// TwinCAT 3 PLC project ErrorTracker
// ProgramVersion: 3.1.4023.0
// libraries:
//   Tc2_Standard, * (Beckhoff Automation GmbH)
//   Tc2_System, * (Beckhoff Automation GmbH)
//   Tc2_Utilities, * (Beckhoff Automation GmbH)
//   Tc3_Module, * (Beckhoff Automation GmbH)
// project tree:
//   Diag/ CheckBounds.TcPOU, CheckDivDInt.TcPOU, CheckDivLInt.TcPOU, CheckDivLReal.TcPOU, CheckDivReal.TcPOU, CheckLRangeSigned.TcPOU, CheckLRangeUnsigned.TcPOU, CheckPointer.TcPOU, CheckRangeSigned.TcPOU, CheckRangeUnsigned.TcPOU, E_ErrType.TcDUT, FB_UdintTrig.TcPOU, G_Diag.TcGVL, prgDiag.TcPOU, stErrType.TcDUT, Visu_Diag.TcVIS
//   / GlobalTextList.TcGTLO, PlcTask.TcTTO, Visualization Manager.TcVMO (not stored)
//   POUs/ MAIN.TcPOU
// real-time tasks:
//   TASK PlcTask: cycle T#10ms, priority 20, ADS port 350
// I/O:
//   DEVICE Device 1 (EtherCAT) (disabled), AmsNetId 5.80.91.146.2.1
//     Term 1 (EK1100) [EK1100 EtherCAT Coupler (2A E-Bus)]
//       Term 2 (EL2008) [EL2008 8Ch. Dig. Output 24V, 0.5A]
// variable links:
//   ErrorTracker/ErrorTracker Instance <-> Device 1 (EtherCAT)
//     PlcTask Inputs/prgDiag.uiECatState <-> Inputs/DevState

CONFIGURATION ErrorTracker
    RESOURCE PLC ON TwinCAT3
        TASK PlcTask(INTERVAL := T#10ms, PRIORITY := 20);
        PROGRAM MAIN WITH PlcTask : MAIN;
    END_RESOURCE
END_CONFIGURATION

// ---- Diag/E_ErrType.TcDUT
{attribute 'qualified_only'}
{attribute 'strict'}
TYPE E_ErrType :
(
	eFirStErr,
	eCheckBoundsErr,
	eCheckDivDint,
	eCheckDivLint,
	eCheckDivReal,
	eCheckRange,
	eCheckPointer,
	eEtherCATErr,
	eRuntimeErr,
	eLastErr
);
END_TYPE

// ---- Diag/stErrType.TcDUT
TYPE stErrType :
STRUCT
	horario:DT;
	eErrType:E_ErrType;
END_STRUCT
END_TYPE

// ---- Diag/G_Diag.TcGVL
{attribute 'qualified_only'}
VAR_GLOBAL PERSISTENT
	uiCheckBound:UDINT;
	uiCheckDivDint:UDINT;
	uiCheckDivLint:UDINT;
	uiCheckDivReal:UDINT;
	uiCheckRange:UDINT;
	uiCheckPointer:UDINT;
	uiErrEtherCAT:UDINT;
	uiRuntimeErr:UDINT;
	aErrList:ARRAY[1..uiMaxNumOfErr] OF stErrType;
	uiECatState:UINT;
END_VAR
VAR_GLOBAL CONSTANT
	uiMaxNumOfErr:UINT:=100;
END_VAR

// ---- POUs/MAIN.TcPOU
PROGRAM MAIN
VAR
	i1,i2:INT;
	i3:INT:=5;
END_VAR
//An UPS is necessary to save the persistent Data, if it's not available other options are also possible, such as:
//Save to retain data / text files/Databases or simple use the FB_WritePersistentData and soon as a new error occur to make sure it's gonna be persistent
//Note : leaving Checks activated on a running machine can have negative effects on the performance
//As you find out what's the problem you should also remove checks from your code

//Here we call the program which handles the diagnosis
//
prgDiag();

i1:=i2/i3;

END_PROGRAM

// ---- Diag/prgDiag.TcPOU
PROGRAM prgDiag
VAR
	aErrTrig:ARRAY[E_ErrType.eFirStErr..E_ErrType.eLastErr] OF FB_UdintTrig;
	taskInfo:PlcTaskSystemInfo;
	
	horaAtual: DT;
	uiECatState AT %I*:UINT;
	localTyme:FB_LocalSystemTime;
	trigECAT:R_TRIG;
	timeStartup: TON := (PT := TIME#2S0MS);
	
END_VAR

timeStartup(IN:= TRUE);

IF NOT timeStartup.Q THEN
	RETURN;
END_IF

localTyme(
	sNetID:= '', 
	bEnable:= TRUE, 
	dwCycle:= , 
	dwOpt:= , 
	tTimeout:= , 
	bValid=> , 
	systemTime=> , 
	tzID=> );


taskInfo := _TaskInfo[1];

aErrTrig[E_ErrType.eCheckBoundsErr](uiIn:=G_Diag.uiCheckBound);
aErrTrig[E_ErrType.eCheckDivDint](uiIn:=G_Diag.uiCheckDivDint);
aErrTrig[E_ErrType.eCheckDivLint](uiIn:=G_Diag.uiCheckDivLint);
aErrTrig[E_ErrType.eCheckDivReal](uiIn:=G_Diag.uiCheckDivReal);
aErrTrig[E_ErrType.eCheckRange](uiIn:=G_Diag.uiCheckRange);
aErrTrig[E_ErrType.eCheckPointer](uiIn:=G_Diag.uiCheckPointer);


horaAtual:=SYSTEMTIME_TO_DT(localTyme.systemTime);	//==> colocar a hora do sistema aqui 
{Region "Checks"}
IF aErrTrig[E_ErrType.eCheckBoundsErr].bOut THEN
	M_InsertOnList(eErrInsert:=E_ErrType.eCheckBoundsErr , hora:=horaAtual );
END_IF
IF aErrTrig[E_ErrType.eCheckDivDint].bOut THEN
	M_InsertOnList(eErrInsert:=E_ErrType.eCheckDivDint , hora:=horaAtual );	
END_IF
IF aErrTrig[E_ErrType.eCheckDivLint].bOut THEN
	M_InsertOnList(eErrInsert:= E_ErrType.eCheckDivLint, hora:=horaAtual );	
END_IF
IF aErrTrig[E_ErrType.eCheckDivReal].bOut THEN
	M_InsertOnList(eErrInsert:= E_ErrType.eCheckDivReal, hora:=horaAtual );	
END_IF
IF aErrTrig[E_ErrType.eCheckRange].bOut THEN
	M_InsertOnList(eErrInsert:=E_ErrType.eCheckRange , hora:=horaAtual );	
END_IF
IF aErrTrig[E_ErrType.eCheckPointer].bOut THEN
	M_InsertOnList(eErrInsert:= E_ErrType.eCheckPointer, hora:=horaAtual );	
END_IF
{endregion}

{Region "EtherCAT"}
	trigECAT(CLK:=uiECatState <> 0);
	IF trigECAT.Q THEN
		 M_InsertOnList(eErrInsert:= E_ErrType.eEtherCATErr, hora:=horaAtual );
		 G_Diag.uiECatState:=uiECatState;
	END_IF
{endregion}

{Region "Runtime"}
	IF taskInfo.CycleTimeExceeded THEN
		G_Diag.uiRuntimeErr:=G_Diag.uiRuntimeErr+1;
		M_InsertOnList(eErrInsert:= E_ErrType.eRuntimeErr, hora:=horaAtual );	
	END_IF
{endregion}

METHOD M_InsertOnList : BOOL
VAR_INPUT
	eErrInsert:E_ErrType;
	hora:DT;
END_VAR

VAR
	i: UINT;
END_VAR
FOR i := 100 TO 2 BY -1 DO
	G_Diag.aErrList[i]:=G_Diag.aErrList[i-1];
END_FOR
G_Diag.aErrList[1].eErrType:=eErrInsert;
G_Diag.aErrList[1].horario:=hora;
END_METHOD

END_PROGRAM

// ---- Diag/FB_UdintTrig.TcPOU
FUNCTION_BLOCK FB_UdintTrig
VAR_INPUT
	uiIn:UDINT;
END_VAR
VAR_OUTPUT
	bOut: BOOL;

END_VAR
VAR
	uiOld:UDINT;
	tAllowNewErr:TON;
	bFirst:BOOL:=TRUE;
END_VAR


bOut:= uiIn <> uiOld AND tAllowNewErr.Q AND NOT bFirst;
tAllowNewErr(IN:=uiIn = uiOld , PT:= T#5S);
uiOld:=uiIn;
bFirst:=FALSE;

END_FUNCTION_BLOCK

// ---- Diag/CheckBounds.TcPOU
// Implicitly generated code : DO NOT EDIT
FUNCTION CheckBounds : DINT
VAR_INPUT
	index, lower, upper: DINT;
END_VAR

// Implicitly generated code : Only an Implementation suggestion
{noflow}
IF  index < lower THEN
	G_Diag.uiCheckBound:=G_Diag.uiCheckBound+1;
	CheckBounds := lower;
ELSIF  index > upper THEN
	G_Diag.uiCheckBound:=G_Diag.uiCheckBound+1;
	CheckBounds := upper;
ELSE
	CheckBounds := index;
END_IF
{flow}

END_FUNCTION

// ---- Diag/CheckDivDInt.TcPOU
// Implicitly generated code : DO NOT EDIT
FUNCTION CheckDivDInt : DINT
VAR_INPUT
	divisor:DINT;
END_VAR

// Implicitly generated code : Only an Implementation suggestion
{noflow}
IF divisor = 0 THEN
	G_Diag.uiCheckDivDint:=G_Diag.uiCheckDivDint+1;
	CheckDivDInt:=1;
ELSE
	CheckDivDInt:=divisor;
END_IF;
{flow}

END_FUNCTION

// ---- Diag/CheckDivLInt.TcPOU
// Implicitly generated code : DO NOT EDIT
FUNCTION CheckDivLInt : LINT
VAR_INPUT
	divisor:LINT;
END_VAR

// Implicitly generated code : Only an Implementation suggestion
{noflow}
IF divisor = 0 THEN
	CheckDivLInt:=1;
	G_Diag.uiCheckDivLint:=G_Diag.uiCheckDivLint+1;
ELSE
	CheckDivLInt:=divisor;
END_IF;
{flow}

END_FUNCTION

// ---- Diag/CheckDivLReal.TcPOU
// Implicitly generated code : DO NOT EDIT
FUNCTION CheckDivLReal : LREAL
VAR_INPUT
	divisor:LREAL;
END_VAR

// Implicitly generated code : Only an Implementation suggestion
{noflow}
IF divisor = 0 THEN
	CheckDivLReal:=1;
	G_Diag.uiCheckDivReal:=G_Diag.uiCheckDivReal+1;
ELSE
	CheckDivLReal:=divisor;
END_IF;
{flow}

END_FUNCTION

// ---- Diag/CheckDivReal.TcPOU
// Implicitly generated code : DO NOT EDIT
FUNCTION CheckDivReal : REAL
VAR_INPUT
	divisor:REAL;
END_VAR

// Implicitly generated code : Only an Implementation suggestion
{noflow}
IF divisor = 0 THEN
	CheckDivReal:=1;
	G_Diag.uiCheckDivReal:=G_Diag.uiCheckDivReal+1;
ELSE
	CheckDivReal:=divisor;
END_IF;
{flow}

END_FUNCTION

// ---- Diag/CheckLRangeSigned.TcPOU
// Implicitly generated code : DO NOT EDIT
FUNCTION CheckLRangeSigned : LINT
VAR_INPUT
	value, lower, upper: LINT;
END_VAR

// Implicitly generated code : Only an Implementation suggestion
{noflow}
IF (value < lower) THEN
	CheckLRangeSigned := lower;
	G_Diag.uiCheckRange:=G_Diag.uiCheckRange+1;
ELSIF(value > upper) THEN
	CheckLRangeSigned := upper;
	G_Diag.uiCheckRange:=G_Diag.uiCheckRange+1;
ELSE
	CheckLRangeSigned := value;
END_IF

{flow}

END_FUNCTION

// ---- Diag/CheckLRangeUnsigned.TcPOU
// Implicitly generated code : DO NOT EDIT
FUNCTION CheckLRangeUnsigned : ULINT
VAR_INPUT
	value, lower, upper: ULINT;
END_VAR

// Implicitly generated code : Only an Implementation suggestion
{noflow}
IF (value < lower) THEN
	CheckLRangeUnsigned := lower;
ELSIF(value > upper) THEN
	CheckLRangeUnsigned := upper;
ELSE
	CheckLRangeUnsigned := value;
END_IF
{flow}

END_FUNCTION

// ---- Diag/CheckPointer.TcPOU
// Implicitly generated code : DO NOT EDIT
FUNCTION CheckPointer : POINTER TO BYTE
VAR_INPUT 
	ptToTest : POINTER TO BYTE; // Destination address of the pointer
	iSize : DINT;		        // Size of the type the pointer points to. (e.g: 20 for POINTER TO ARRAY [0..9] OF INT) 
	iGran : DINT;		        // Granularity of the pointer access. This is the size of the biggest non-structured data type in the type the pointer points to. (e.g: 2 for POINTER TO ARRAY [0..9] OF INT)
	bWrite: BOOL;		        // Indicates read or write Access. TRUE = write access.
END_VAR

// No standard way of implementation. Fill your own code here
CheckPointer := ptToTest;

G_Diag.uiCheckPointer:=G_Diag.uiCheckPointer+1;
{flow}

END_FUNCTION

// ---- Diag/CheckRangeSigned.TcPOU
// Implicitly generated code : DO NOT EDIT
FUNCTION CheckRangeSigned : DINT
VAR_INPUT
	value, lower, upper: DINT;
END_VAR

// Implicitly generated code : Only an Implementation suggestion
{noflow}
IF (value < lower) THEN
	CheckRangeSigned := lower;
	G_Diag.uiCheckRange:=G_Diag.uiCheckRange+1;
ELSIF(value > upper) THEN
	CheckRangeSigned := upper;
	G_Diag.uiCheckRange:=G_Diag.uiCheckRange+1;
ELSE
	CheckRangeSigned := value;
END_IF
{flow}

END_FUNCTION

// ---- Diag/CheckRangeUnsigned.TcPOU
// Implicitly generated code : DO NOT EDIT
FUNCTION CheckRangeUnsigned : UDINT
VAR_INPUT
	value, lower, upper: UDINT;
END_VAR

// Implicitly generated code : Only an Implementation suggestion
{noflow}
IF (value < lower) THEN
	CheckRangeUnsigned := lower;
	G_Diag.uiCheckRange:=G_Diag.uiCheckRange+1;
ELSIF(value > upper) THEN
	CheckRangeUnsigned := upper;
	G_Diag.uiCheckRange:=G_Diag.uiCheckRange+1;
ELSE
	CheckRangeUnsigned := value;
END_IF
{flow}

END_FUNCTION

// ---- Diag/Visu_Diag.TcVIS
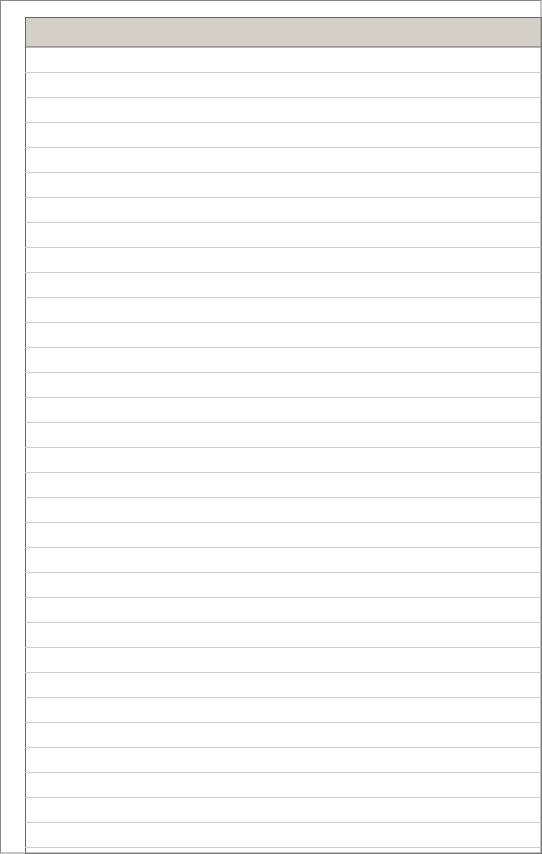
VISUALIZATION Visu_Diag  // 542x854
    Table (25,17 517x837), data array: G_Diag.aErrList
        p3854506369: G_Diag.aErrList[INDEX].horario
        p1892666644: G_Diag.aErrList[INDEX].eErrType
        p2232123230: Timestamp
        p511219082: Eror Type
END_VISUALIZATION

// ---- GlobalTextList.TcGTLO
TEXTLIST GlobalTextList
  435 = 'Eror Type'
  340 = 'Horario'
  200 = 'Timestamp'
  341 = 'Tipo do erro'
END_TEXTLIST
